(* CoDeSys 2.3 project: Sample04.pro *)
(* Libraries: STANDARD.LIB 5.6.98 10:31:02 *)

(* Task configuration *)
TASK Standard (PRIORITY := 0, INTERVAL := T#10ms);
	MAIN
END_TASK

(* POU MAIN, ST *)
PROGRAM MAIN
VAR
	text : STRING[30] := 'hello';
END_VAR
;
END_PROGRAM
